TYPE TYP_RYG_TOWER_HW :
STRUCT
	Out : TYP_RYG_TOWER_HW_OUT;
END_STRUCT
END_TYPE

(* stored: Version 1.1.0.1, ProductVersion 3.1.4024.12
   DUT TYP_RYG_TOWER_HW: Id {f26081aa-e192-4e86-9052-2c5b0ddc79a1} *)
